FUNCTION_BLOCK TIME_Param
VAR_INPUT PERSISTENT
	val			: TIME;
END_VAR

END_FUNCTION_BLOCK

(* stored: Version 1.1.0.1
   POU TIME_Param: Id {ab52f2c8-822a-4785-a83d-b1c5010eebf1}, SpecialFunc None *)
